% RSLogix 500 project HEATER.RSS, saved by version 9.00.00.04 %
PROJECT "UNTITLED"    % processor: Bul.1763 MicroLogix 1100 Series A %

PROGRAM FILES
  LAD 2   6 rungs

DATA FILES
  O0 OUTPUT  9 elements
  I1 INPUT  16 elements
  S2 STATUS  66 elements
  B3 BINARY  1 elements
  T4 TIMER  1 elements
  C5 COUNTER  1 elements
  R6 CONTROL  1 elements
  N7 INTEGER  2 elements
  F8 FLOAT  1 elements
  PD9 TEMP  1 elements

LADDER 2
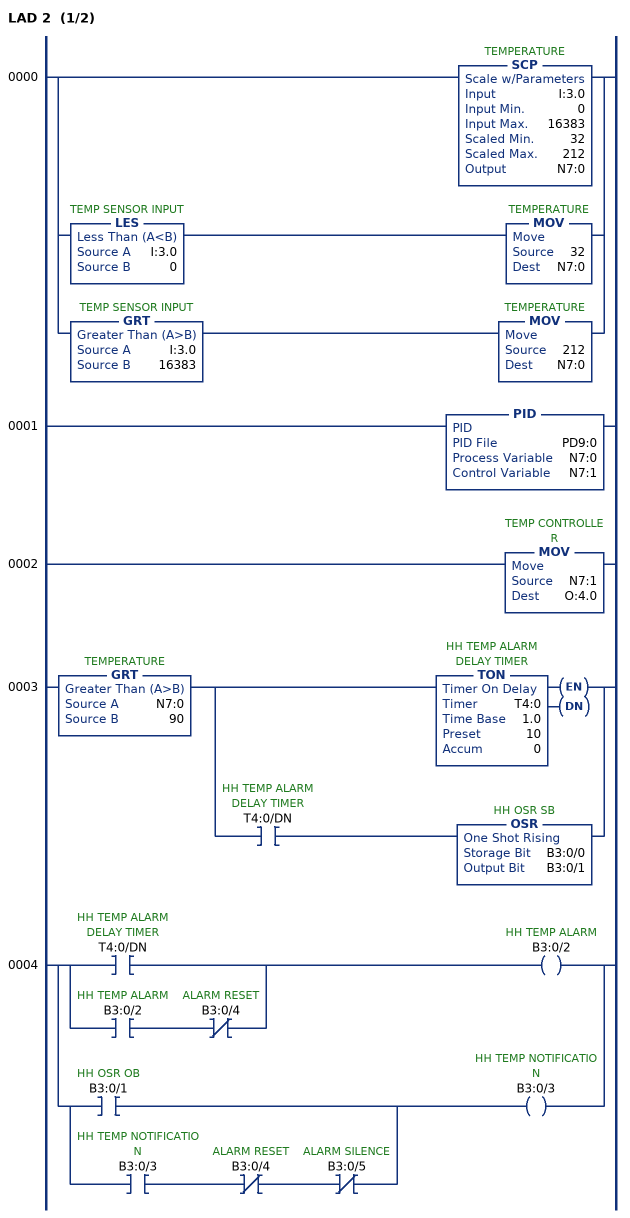
% Rung: 0 %
SOR BST SCP I:3.0 0 16383 32 212 N7:0 NXB LES I:3.0 0 MOV 32 N7:0 NXB GRT I:3.0 16383 MOV 212 N7:0 BND EOR
%   I:3.0  "TEMP SENSOR INPUT" %
%   N7:0  "TEMPERATURE" %
% Rung: 1 %
SOR PID PD9:0 N7:0 N7:1 EOR
%   N7:0  "TEMPERATURE" %
%   N7:1  "PID OUTPUT" %
% Rung: 2 %
SOR MOV N7:1 O:4.0 EOR
%   N7:1  "PID OUTPUT" %
%   O:4.0  "TEMP CONTROLLER" %
% Rung: 3 %
SOR GRT N7:0 90 BST TON T4:0 1.0 10 0 NXB XIC T4:0/DN OSR B3:0/0 B3:0/1 BND EOR
%   N7:0  "TEMPERATURE" %
%   T4:0  "HH TEMP ALARM DELAY TIMER" %
%   B3:0/0  "HH OSR SB" %
%   B3:0/1  "HH OSR OB" %
% Rung: 4 %
SOR BST BST XIC T4:0/DN NXB XIC B3:0/2 XIO B3:0/4 BND OTE B3:0/2 NXB BST XIC B3:0/1 NXB XIC B3:0/3 XIO B3:0/4 XIO B3:0/5 BND OTE B3:0/3 BND EOR
%   T4:0  "HH TEMP ALARM DELAY TIMER" %
%   B3:0/2  "HH TEMP ALARM" %
%   B3:0/4  "ALARM RESET" %
%   B3:0/1  "HH OSR OB" %
%   B3:0/3  "HH TEMP NOTIFICATION" %
%   B3:0/5  "ALARM SILENCE" %

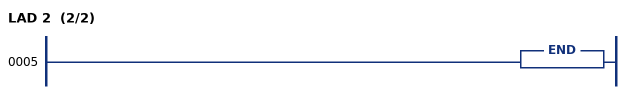
% Rung: 5 %
SOR END EOR

OTHER DOCUMENTED ADDRESSES
  I:1.0/0  "LOW TEMP SWITCH INPUT"
  I:1.0/1  "HIGH SWITCH INPUT"
  O:2.0/0  "HEATER OUTPUT"

DATA TABLE (non-zero values as saved)
DATA T4
% .PRE .ACC %
% T4:0 % 10 0
